FUNCTION_BLOCK Test_TStreamAdd_Read_UDINT EXTENDS T_UnitTestBase
VAR
    Stream  : T_Stream(StreamLength := 2);
    ArgType : E_ArgTypeId := E_ArgTypeId.Type_UDINT;
END_VAR

Stream.Init(2);

// add a UDINT...
Stream.SetNextArgTypeId(ArgType);
Stream.Add_UDINT(12345678);

Stream.SetReadPosition(0);

// check next arg type is correct...
Assertion.AssertEquals_INT(Expected     := ArgType,
                           Actual       := Stream.GetNextArgTypeId(),
                           VariableName := 'Stream.GetNextArgTypeId()');

// check next value...	
Assertion.AssertEquals_UDINT(Expected     := 12345678,
                             Actual       := Stream.Read_UDINT(),
                             VariableName := 'Stream.Read_UDINT()');

// check we are at the end of the stream..							
Assertion.AssertEquals_UDINT(Expected     := Stream.StreamLength,
                             Actual       := Stream.ReadPosition,
                             VariableName := 'Stream.ReadPosition');

TestFinished();

END_FUNCTION_BLOCK

(* stored: Version 1.1.0.1, ProductVersion 3.1.4024.9
   POU Test_TStreamAdd_Read_UDINT: Id {1ea943e2-a807-4204-9494-af8b2ba37d4b}, SpecialFunc None *)
